DATA_BLOCK "dbArchiveControlOven"
{ S7_Optimized_Access := 'TRUE' }
VERSION : 0.8
NON_RETAIN
"fbArchiveControlOven"

BEGIN

END_DATA_BLOCK

